FUNCTION_BLOCK CLICK_CNT
VAR_INPUT
	IN : BOOL;
	N : INT;
	TC : TIME;
END_VAR
VAR_OUTPUT
	Q : BOOL;
END_VAR
VAR
	tx : TP;
	edge: BOOL;
	cnt: INT := -1;
END_VAR

(*
version 1.0	16. jul. 2008
programmer 	hugo
tested by	oscat

this Module decodes a specified number of clicks.
the output trig is high for one cycle if N clicks are present within a specified time TC.

*)

(* Q shall only be active for one cycle only *)
Q := FALSE;

IF in AND NOT edge AND NOT tx.q THEN
	(* a rising edge on in sets the counter to 0 *)
	cnt := 0;
ELSIF tx.Q AND NOT IN AND edge THEN
	(* count falling edges when tp.q is true *)
	cnt := cnt + 1;
ELSIF NOT tx.Q THEN
	Q := cnt = N;
	cnt := -1;
END_IF;

(* remember the status of IN *)
edge := IN;
tx(in := IN, pt := TC);


(* revision history

hm 	16. jul. 2008	rev 1.0
	original version released


*)

END_FUNCTION_BLOCK

(* stored: Version 1.1.0.1, ProductVersion 3.1.4022.7
   POU CLICK_CNT: Id {ede6bdf2-2a74-48b0-b416-7cff12d5f199}, SpecialFunc None *)
